// TIA Portal project "Clasificación, llenado y tapado de envases de pintura" (V16)

(* hardware
DEVICE "S7300/ET200M station_1"  S7-300 station
   slot 0: "Rail_0"  Rail  6ES7 390-1***0-0AA0
   slot 2: "PLC_1"  CPU 314C-2 PN/DP  6ES7 314-6EH04-0AB0  V3.3
      slot 2: "PROFINET interface_1"  PN-IO
         slot 1: "Port_1"  Port
         slot 2: "Port_2"  Port
      slot 5: "DI 24/DO 16_1"  DI24/DO16
      slot 6: "AI 5/AO 2_1"  AI5/AO2
      slot 7: "Count_1"  Counter
      slot 8: "Positioning_1"  Positioning
DEVICE "HMI_1"  TP700 Comfort
   slot 0: "HMI_1"  TP700 Comfort  6AV2 124-0GC01-0AX0  16.0.0.0
   slot 1: "HMI_RT_1"  TP700 Comfort  6AV2 124-0GC01-0AX0  16.0.0.0
   slot 5: "HMI_1.IE_CP_1"  PROFINET Interface  16.0.0.0
      slot 1: "Interfaz PROFINET_1"  PROFINET Interface
         slot 1: "Port_1"  Port
         slot 2: "Port_2"  Port
   slot 7: "HMI_1.MPI/DP_CP_1"  MPI/DP Interface  16.0.0.0
*)

// ===== PLC "PLC_1"  CPU 314C-2 PN/DP =====

VAR_GLOBAL   // PLC tag table "Entradas"
   "START" AT %I0.0 : Bool;
   "STOP" AT %I0.1 : Bool;
   "SPosIzq1" AT %I0.2 : Bool;
   "SPosDer1" AT %I0.3 : Bool;
   "PE" AT %I0.4 : Bool;
   "SVision" AT %ID30 : DInt;
   "SPosDer2" AT %I0.5 : Bool;
   "SPoseDer3" AT %I0.6 : Bool;
   "SPosIzq2" AT %I0.7 : Bool;
   "SPosIzq3" AT %I1.0 : Bool;
   "SEntrada" AT %I1.1 : Bool;
   "START_HMI" AT %M3.7 : Bool;
   "STOP_HMI" AT %M4.0 : Bool;
   "PE_HMI" AT %M4.1 : Bool;
   "EnvAzul" AT %M4.2 : Bool;
   "EnvVerde" AT %M4.3 : Bool;
   "SPosIzq4" AT %I1.2 : Bool;
   "SPosDer4" AT %I1.3 : Bool;
   "ContadorEnvAzul" AT %MW0 : Int;
   "ContadorEnvVerd" AT %MW2 : Int;
   "ClasificadorRecto" AT %M4.4 : Bool;
   "SEntTapaAzul" AT %I1.4 : Bool;
   "SEntTapaVerd" AT %I1.5 : Bool;
END_VAR

VAR_GLOBAL   // PLC tag table "Salidas"
   "FajaEntr" AT %Q0.0 : Bool;
   "ClasificadorGiro" AT %Q0.1 : Bool;
   "ClasificadorFaja+" AT %Q0.2 : Bool;
   "VLlenTanqIzq" AT %Q0.3 : Bool;
   "VLlenTanqDer" AT %Q0.4 : Bool;
   "FajaIzq1" AT %Q0.5 : Bool;
   "FajaIzq2" AT %Q0.6 : Bool;
   "FajaIzq3" AT %Q0.7 : Bool;
   "VLlenadoEnvIzq" AT %Q1.0 : Bool;
   "VDescTanqIzq" AT %Q1.1 : Bool;
   "FajaDer1" AT %Q1.2 : Bool;
   "VLlenadoEnvDer" AT %Q1.3 : Bool;
   "VDescTanqDer" AT %Q1.4 : Bool;
   "FajaDerecha2" AT %Q1.5 : Bool;
   "FajaDerecha3" AT %Q1.6 : Bool;
   "FajaIzq4" AT %Q1.7 : Bool;
   "FajaIzq5" AT %Q2.0 : Bool;
   "ClampDere1" AT %Q2.1 : Bool;
   "RaiseDere" AT %Q2.2 : Bool;
   "ClampDere2" AT %Q2.3 : Bool;
   "ClampIzq1" AT %Q2.4 : Bool;
   "RaiseIzq" AT %Q2.5 : Bool;
   "ClampIzq2" AT %Q2.6 : Bool;
   "MovZRDer" AT %Q2.7 : Bool;
   "MovXRder" AT %Q3.0 : Bool;
   "GrabRDer" AT %Q3.1 : Bool;
   "MovZRIzq" AT %Q3.2 : Bool;
   "MovXRizq" AT %Q3.3 : Bool;
   "GrabRIzq" AT %Q3.4 : Bool;
END_VAR

VAR_GLOBAL   // PLC tag table "Memorias"
   "Operativo" AT %M5.0 : Bool;
   "Tem1" AT %M0.1 : Bool;
   "Tem2" AT %M0.2 : Bool;
   "Tem3" AT %M0.3 : Bool;
   "Tem4" AT %M0.4 : Bool;
   "Tem6" AT %M0.6 : Bool;
   "Tem7" AT %M0.7 : Bool;
   "Tem8" AT %M1.0 : Bool;
   "Tem9" AT %M1.1 : Bool;
   "Tem10" AT %M1.2 : Bool;
   "Tem11" AT %M1.3 : Bool;
   "Tem12" AT %M1.4 : Bool;
   "Tem13" AT %M1.5 : Bool;
   "Tem14" AT %M1.6 : Bool;
   "Tem15" AT %M1.7 : Bool;
   "Tem16" AT %M2.0 : Bool;
   "Tem17" AT %M2.1 : Bool;
   "Tem18" AT %M2.2 : Bool;
   "Tem19" AT %M2.3 : Bool;
   "Tem20" AT %M2.4 : Bool;
   "Tem21" AT %M2.5 : Bool;
   "Tem22" AT %M2.6 : Bool;
   "Tem23" AT %M2.7 : Bool;
   "Tem24" AT %M3.0 : Bool;
   "Tem25" AT %M3.1 : Bool;
   "Tem26" AT %M3.2 : Bool;
   "Tem27" AT %M3.3 : Bool;
   "Tem28" AT %M3.4 : Bool;
   "Tem29" AT %M3.5 : Bool;
   "Tem30" AT %M3.6 : Bool;
END_VAR

DATA_BLOCK "Block_1_DB"   // DB1
{ S7_Optimized_Access := 'FALSE' }
VERSION : 0.1
// stored: InstanceOfName Block_1
"Block_1"
BEGIN
END_DATA_BLOCK

FUNCTION_BLOCK "Block_1"   // FB1, GRAPH
{ S7_Optimized_Access := 'FALSE' }
VERSION : 0.1
   VAR_INPUT
      OFF_SQ : Bool := false;   // Turn sequence off
      INIT_SQ : Bool := false;   // Set sequence to initial state
      ACK_EF : Bool := false;   // Acknowledge all errors and faults
      S_PREV : Bool := false;   // Output previous step in parameter S_NO
      S_NEXT : Bool := false;   // Indicate next step in parameter S_NO
      SW_AUTO : Bool := false;   // Automatic mode
      SW_TAP : Bool := false;   // Semiautomatic/switch with transition
      SW_TOP : Bool := false;   // Semiautomatic/ignore transition
      SW_MAN : Bool := false;   // Manual mode
      S_SEL : Int := 0;   // Select step to be output to S_NO
      S_ON : Bool := false;   // Activate step indicated in S_NO
      S_OFF : Bool := false;   // Deactivate step indicated S_NO
      T_PUSH : Bool := false;   // Enable transition to switch in semi automatic mode
   END_VAR
   VAR_OUTPUT
      S_NO : Int := 0;   // Step number
      S_MORE : Bool := false;   // More steps are available and can be shown in S_NO
      S_ACTIVE : Bool := false;   // Step indicated in S_NO is active
      ERR_FLT : Bool := false;   // Interlock or supervision group error
      AUTO_ON : Bool := false;   // Automatic mode is active
      TAP_ON : Bool := false;   // Semiautomatic mode/step with transition enabled
      TOP_ON : Bool := false;   // Semiautomatic mode/ignore transition enabled
      MAN_ON : Bool := false;   // Manual mode is active
   END_VAR
   VAR
      SWITCH : Array[0..2] of DWord;
      SW_SQTS : Array[0..36] of Byte;
      SW_ADDR : Word := 16#A;
      G7T_0 : GraphTransition;
      G7S_0 : GraphStep;
      PRE_CRIT : Array[0..0] of DWord;
      POST_CRIT : Array[0..0] of DWord;
      TVX : Array[0..8] of Byte;
      TTX : Array[0..8] of Byte;
      TSX : Array[0..6] of Byte;
      S00X : Array[0..6] of Byte;
      SOFFX : Array[0..6] of Byte;
      SONX : Array[0..6] of Byte;
      SAX : Array[0..6] of Byte;
      SERRX : Array[0..37] of Byte;
      SMX : Array[0..37] of Byte;
      S0X : Array[0..37] of Byte;
      S1X : Array[0..37] of Byte;
      S_DISPLAY : Int;   // Internal display of output parameter S_NO
      S_SEL_OLD : Int;   // Previous value in S_SEL
      S_DISPIDX : Byte;   // Index of the step in S_NO
      T_DISPIDX : Byte;   // Index of the transition displayed in T_NO
      MOPEDGE : Struct
         AUTO : Bool := false;
         MAN : Bool := false;
         TAP : Bool := false;
         TOP : Bool := false;
         ACK_S : Bool := false;
         REG_S : Bool := false;
         T_PREV : Bool := false;
         T_NEXT : Bool := false;
         LOCK : Bool := false;
         SUP : Bool := false;
         ACKREQ : Bool := false;
         SSKIP : Bool := false;
         OFF : Bool := false;
         INIT : Bool := false;
         HALT : Bool := false;
         TMS_HALT : Bool := false;
         OPS_ZERO : Bool := false;
         SACT_DISP : Bool := false;
         SEF_DISP : Bool := false;
         SALL_DISP : Bool := false;
         S_PREV : Bool := false;
         S_NEXT : Bool := false;
         S_SELOK : Bool := false;
         S_ON : Bool := false;
         S_OFF : Bool := false;
         T_PUSH : Bool := false;
         REG : Bool := false;
         ACK : Bool := false;
         IL_PERM : Bool := false;
         T_PERM : Bool := false;
         ILP_MAN : Bool := false;
      END_STRUCT;
      MOP : Struct   // Mode
         AUTO : Bool := true;   // Status: automatic mode
         MAN : Bool := false;   // Status: manual mode
         TAP : Bool := false;   // Status: semi automatic/switch with transition
         TOP : Bool := false;   // Status: semi automatic/ignore transition
         ACK_S : Bool := false;   // Request: acknowledge step at parameter S_NO
         REG_S : Bool := false;   // Request: register step indicated in S_NO
         T_PREV : Bool := false;   // Request: output previous valid transition in T_NO
         T_NEXT : Bool := false;   // Request: output next valid transition in T_NO
         LOCK : Bool := true;   // Status: interlocks activated
         SUP : Bool := true;   // Status: supervisions activated
         ACKREQ : Bool := true;   // Status: acknowledgment required
         SSKIP : Bool := false;   // Status: "Skip steps" enabled
         OFF : Bool := false;   // Request: deactivate all steps
         INIT : Bool := true;   // Request: set sequence to initial state
         HALT : Bool := false;   // Status: sequence halted
         TMS_HALT : Bool := false;   // Status: all internal timers held
         OPS_ZERO : Bool := false;   // Status: set all operands processed with N, L, D instructions to 0
         SACT_DISP : Bool := true;   // Status: display active steps only
         SEF_DISP : Bool := false;   // Status: display only steps with errors and disrupted steps
         SALL_DISP : Bool := false;   // Status: display all steps
         S_PREV : Bool := false;   // Request: output previous step to S_NO
         S_NEXT : Bool := false;   // Request: Output next step at S_NO parameter
         S_SELOK : Bool := false;   // Request: output step number from S_SEL to S_NO
         S_ON : Bool := false;   // Request: activate step indicated in S_NO
         S_OFF : Bool := false;   // Request: deactivate step at parameter S_NO
         T_PUSH : Bool := false;   // Request: transition switching enabled
         REG : Bool := false;   // Request: register all interlock and supervision errors
         ACK : Bool := false;   // Request: acknowledge all interlock and supervision errors
         IL_PERM : Bool := false;   // Status: permanent processing of all interlocks
         T_PERM : Bool := false;   // Status: permanent processing of all transitions
         ILP_MAN : Bool := false;   // Status: permanent processing of all interlocks in manual mode
      END_STRUCT;
      TICKS : Struct   // Clock speeds
         DELTA : Time := T#0ms;   // Time difference between cycles
         OLD : Time := T#0ms;   // 10 ms clock counter value in last cycle
         NEW : Time := T#0ms;   // 10 ms clock counter value in this cycle
      END_STRUCT;
      SQ_FLAGS : Struct   // Sequence bit memory
         ERR_FLT : Bool := false;   // Interlock and supervision group error
         ERROR : Bool := false;   // Interlock group error
         FAULT : Bool := false;   // Supervision group error
         RT_FAIL : Bool := false;   // Runtime error
         NO_SNO : Bool := false;   // Requested step number not found
         NF_OFL : Bool := false;   // Overflow: too many ON or OFF requests
         SA_OFL : Bool := false;   // Overflow: too many steps active
         TV_OFL : Bool := false;   // Overflow: too many valid transitions
         MSG_OFL : Bool := false;   // Overflow: not enough system resources for ALARM_S
         NO_SWI : Bool := false;   // Do not switch in this cycle
         CYC_OP : Bool := false;   // Cyclic execution of the sequence after initialization
         AS_MSG : Bool := true;   // Alarms during runtime enabled or disabled by instruction
         AS_SEND : Bool := false;   // Send alarms from WR_USMSG or only enter in diagnostics buffer
         SQ_BUSY : Bool := false;   // Internal edge memory bit for sequence processing
         SA_BUSY : Bool := false;   // Internal edge memory bit for sequence processing
         AS_SIG : Bool := false;   // Edge memory bit for alarms from Alarm_S and Alarm_SQ
      END_STRUCT;
      S_PTR : DWord := 16#13F0;
      S_PTR2 : DWord := 16#0;
      S_PTR3 : DWord := 16#3EA0;
      S_PTR4 : DWord := 16#3D70;
      T_PTR : DWord := 16#3C40;
      C_AR2 : DWord := 16#0;
      M_FBDB : DWord := 16#10000;
      M_SNO : Word := 16#0;
      M_EVID : Word := 16#0;
      M_EVIL : C_Alarm_s;
      M_EVSV : C_Alarm_s;
      M_EV : DWord := 16#3A50;
      CRIT : Array[0..31] of Bool;
      S_START : Byte := 16#0;
      S_IDX : Byte := 16#0;
      S_INT : Int := 72;
      S_TMP : Byte := 16#0;
      T_START : Byte := 16#0;
      T_IDX : Byte := 16#0;
      T_TMP : Byte := 16#0;
      T_TMP2 : Byte := 16#00;
      TV_POT : Byte := 16#06;
      RETURN1 : Byte := 16#0;
      RETURN2 : Byte := 16#0;
      SINI : Array[0..6] of Byte;
      LSTT : Array[0..35] of Byte;
      ATAJ : Array[0..35] of Byte;
      ATAB : Array[0..35] of Byte;
      PSTT : Array[0..35] of Byte;
      NSTT : Array[0..35] of Byte;
      ASSJ : Array[0..36] of Byte;
      ASSB : Array[0..36] of Byte;
      PTTS : Array[0..36] of Byte;
      NTTS : Array[0..36] of Byte;
      PRE_CNT : Word := 16#1;
      POST_CNT : Word := 16#1;
      ADR_COND : Word := 16#0;
      MAX_TVAL : Byte := 16#7;
      MAX_SACT : Byte := 16#5;
      MAX_CRIT : Byte := 16#4;
      T_CNT : Byte := 16#23;
      SUP_CNT : Byte := 16#0;
      LOCK_CNT : Byte := 16#0;
      S_CNT : Byte := 16#24;
      SQ_CNT : Byte := 16#1;
      PRS_INPAR : DWord := 16#E000FEC8;
      PRS_OUTPAR : DWord := 16#E000800F;
      GC_FLAGS : Struct
         T_MACH : Byte := 16#EB;
         COND_ED : Byte := 16#E3;
         W_LEVEL : Byte := 16#D5;
         FB_IF : Byte := 16#FA;
         AS_MSG : Word := 16#404;
         SSB : Word := 16#108;
         DILG : Word := 16#9CE;
         ADDR_T0 : Word := 16#3E;
         CRIT_AVAIL : Bool := false;
         SSKIP_AVAIL : Bool := true;
         SSKIP_ON : Bool := false;
         ACK_REQ : Bool := true;
         SYNC_AVAIL : Bool := true;
         ILP_MAN : Bool := false;
         SWM_LOCKED : Bool := false;
         SAVE_SW : Bool := true;
      END_STRUCT;
      G7_FBMARK : Byte := 16#3C;
      G7_RELEASE : Byte := 16#3C;
      G7_ID2 : Byte := 16#37;
      G7_ID1 : Byte := 16#47;
   END_VAR
   // SWITCH[0] := 16#2020;
   // SWITCH[1] := 16#20;
   // SWITCH[2] := 16#20000000;
   // SW_SQTS[0] := 16#9;
   // SW_SQTS[4] := 16#1;
   // SW_SQTS[5] := 16#1;
   // SW_SQTS[6] := 16#1;
   // SW_SQTS[7] := 16#1;
   // SW_SQTS[8] := 16#2;
   // SW_SQTS[9] := 16#3;
   // SW_SQTS[10] := 16#2;
   // SW_SQTS[11] := 16#2;
   // SW_SQTS[12] := 16#2;
   // SW_SQTS[13] := 16#2;
   // SW_SQTS[14] := 16#2;
   // SW_SQTS[15] := 16#2;
   // SW_SQTS[16] := 16#2;
   // SW_SQTS[17] := 16#3;
   // SW_SQTS[18] := 16#4;
   // SW_SQTS[19] := 16#5;
   // SW_SQTS[20] := 16#5;
   // SW_SQTS[21] := 16#5;
   // SW_SQTS[22] := 16#5;
   // SW_SQTS[23] := 16#5;
   // SW_SQTS[24] := 16#5;
   // SW_SQTS[25] := 16#6;
   // SW_SQTS[26] := 16#7;
   // SW_SQTS[27] := 16#7;
   // SW_SQTS[28] := 16#6;
   // SW_SQTS[29] := 16#6;
   // SW_SQTS[30] := 16#6;
   // SW_SQTS[31] := 16#6;
   // SW_SQTS[32] := 16#6;
   // SW_SQTS[33] := 16#6;
   // SW_SQTS[34] := 16#6;
   // SW_SQTS[35] := 16#8;
   // SW_SQTS[36] := 16#1;
   // TVX[0] := 16#1;
   // TTX[0] := 16#1;
   // TSX[0] := 16#1;
   // S00X[0] := 16#1;
   // SOFFX[0] := 16#1;
   // SONX[0] := 16#1;
   // SAX[0] := 16#1;
   // SERRX[0] := 16#1;
   // SMX[0] := 16#1;
   // S0X[0] := 16#1;
   // S1X[0] := 16#1;
   // SINI[0] := 16#2;
   // SINI[1] := 16#1;
   // SINI[2] := 0;
   // SINI[3] := 0;
   // SINI[4] := 0;
   // SINI[5] := 0;
   // SINI[6] := 0;
   // LSTT[0] := 0;
   // LSTT[1] := 0;
   // LSTT[2] := 0;
   // LSTT[3] := 0;
   // LSTT[4] := 0;
   // LSTT[5] := 0;
   // LSTT[6] := 0;
   // LSTT[7] := 0;
   // LSTT[8] := 0;
   // LSTT[9] := 0;
   // LSTT[10] := 0;
   // LSTT[11] := 0;
   // LSTT[12] := 0;
   // LSTT[13] := 0;
   // LSTT[14] := 0;
   // LSTT[15] := 0;
   // LSTT[16] := 0;
   // LSTT[17] := 0;
   // LSTT[18] := 0;
   // LSTT[19] := 16#1;
   // LSTT[20] := 0;
   // LSTT[21] := 0;
   // LSTT[22] := 0;
   // LSTT[23] := 0;
   // LSTT[24] := 0;
   // LSTT[25] := 0;
   // LSTT[26] := 0;
   // LSTT[27] := 0;
   // LSTT[28] := 0;
   // LSTT[29] := 0;
   // LSTT[30] := 0;
   // LSTT[31] := 0;
   // LSTT[32] := 0;
   // LSTT[33] := 0;
   // LSTT[34] := 0;
   // LSTT[35] := 16#1;
   // ATAJ[0] := 0;
   // ATAJ[1] := 16#1;
   // ATAJ[2] := 16#2;
   // ATAJ[3] := 16#3;
   // ATAJ[4] := 16#4;
   // ATAJ[5] := 16#5;
   // ATAJ[6] := 16#6;
   // ATAJ[7] := 16#7;
   // ATAJ[8] := 16#8;
   // ATAJ[9] := 16#9;
   // ATAJ[10] := 16#A;
   // ATAJ[11] := 16#B;
   // ATAJ[12] := 16#C;
   // ATAJ[13] := 16#D;
   // ATAJ[14] := 16#E;
   // ATAJ[15] := 16#F;
   // ATAJ[16] := 16#10;
   // ATAJ[17] := 16#11;
   // ATAJ[18] := 16#12;
   // ATAJ[19] := 16#13;
   // ATAJ[20] := 16#14;
   // ATAJ[21] := 16#15;
   // ATAJ[22] := 16#16;
   // ATAJ[23] := 16#17;
   // ATAJ[24] := 16#18;
   // ATAJ[25] := 16#19;
   // ATAJ[26] := 16#1A;
   // ATAJ[27] := 16#1B;
   // ATAJ[28] := 16#1C;
   // ATAJ[29] := 16#1D;
   // ATAJ[30] := 16#1E;
   // ATAJ[31] := 16#1F;
   // ATAJ[32] := 16#20;
   // ATAJ[33] := 16#21;
   // ATAJ[34] := 16#22;
   // ATAJ[35] := 16#23;
   // ATAB[0] := 0;
   // ATAB[1] := 16#1;
   // ATAB[2] := 16#2;
   // ATAB[3] := 16#4;
   // ATAB[4] := 16#3;
   // ATAB[5] := 16#5;
   // ATAB[6] := 16#6;
   // ATAB[7] := 16#7;
   // ATAB[8] := 16#8;
   // ATAB[9] := 16#9;
   // ATAB[10] := 16#A;
   // ATAB[11] := 16#B;
   // ATAB[12] := 16#C;
   // ATAB[13] := 16#D;
   // ATAB[14] := 16#E;
   // ATAB[15] := 16#F;
   // ATAB[16] := 16#10;
   // ATAB[17] := 16#11;
   // ATAB[18] := 16#12;
   // ATAB[19] := 16#13;
   // ATAB[20] := 16#14;
   // ATAB[21] := 16#15;
   // ATAB[22] := 16#16;
   // ATAB[23] := 16#17;
   // ATAB[24] := 16#18;
   // ATAB[25] := 16#19;
   // ATAB[26] := 16#1A;
   // ATAB[27] := 16#1B;
   // ATAB[28] := 16#1C;
   // ATAB[29] := 16#1D;
   // ATAB[30] := 16#1E;
   // ATAB[31] := 16#1F;
   // ATAB[32] := 16#20;
   // ATAB[33] := 16#21;
   // ATAB[34] := 16#22;
   // ATAB[35] := 16#23;
   // PSTT[0] := 0;
   // PSTT[1] := 16#1;
   // PSTT[2] := 16#2;
   // PSTT[3] := 16#3;
   // PSTT[4] := 16#3;
   // PSTT[5] := 16#4;
   // PSTT[6] := 16#5;
   // PSTT[7] := 16#6;
   // PSTT[8] := 16#7;
   // PSTT[9] := 16#24;
   // PSTT[10] := 16#9;
   // PSTT[11] := 16#8;
   // PSTT[12] := 16#A;
   // PSTT[13] := 16#B;
   // PSTT[14] := 16#C;
   // PSTT[15] := 16#D;
   // PSTT[16] := 16#E;
   // PSTT[17] := 16#F;
   // PSTT[18] := 16#11;
   // PSTT[19] := 16#12;
   // PSTT[20] := 16#13;
   // PSTT[21] := 16#14;
   // PSTT[22] := 16#15;
   // PSTT[23] := 16#16;
   // PSTT[24] := 16#17;
   // PSTT[25] := 16#18;
   // PSTT[26] := 16#1A;
   // PSTT[27] := 16#19;
   // PSTT[28] := 16#1C;
   // PSTT[29] := 16#1D;
   // PSTT[30] := 16#1E;
   // PSTT[31] := 16#1F;
   // PSTT[32] := 16#20;
   // PSTT[33] := 16#21;
   // PSTT[34] := 16#1B;
   // PSTT[35] := 16#23;
   // NSTT[0] := 16#1;
   // NSTT[1] := 16#2;
   // NSTT[2] := 16#3;
   // NSTT[3] := 16#13;
   // NSTT[4] := 16#4;
   // NSTT[5] := 16#5;
   // NSTT[6] := 16#6;
   // NSTT[7] := 16#7;
   // NSTT[8] := 16#24;
   // NSTT[9] := 16#9;
   // NSTT[10] := 16#11;
   // NSTT[11] := 16#A;
   // NSTT[12] := 16#B;
   // NSTT[13] := 16#C;
   // NSTT[14] := 16#D;
   // NSTT[15] := 16#E;
   // NSTT[16] := 16#F;
   // NSTT[17] := 16#10;
   // NSTT[18] := 16#12;
   // NSTT[19] := 16#1;
   // NSTT[20] := 16#14;
   // NSTT[21] := 16#15;
   // NSTT[22] := 16#16;
   // NSTT[23] := 16#17;
   // NSTT[24] := 16#18;
   // NSTT[25] := 16#1A;
   // NSTT[26] := 16#1B;
   // NSTT[27] := 16#1C;
   // NSTT[28] := 16#1D;
   // NSTT[29] := 16#1E;
   // NSTT[30] := 16#1F;
   // NSTT[31] := 16#20;
   // NSTT[32] := 16#21;
   // NSTT[33] := 16#22;
   // NSTT[34] := 16#23;
   // NSTT[35] := 16#1;
   // ASSJ[0] := 0;
   // ASSJ[1] := 16#1;
   // ASSJ[2] := 16#2;
   // ASSJ[3] := 16#3;
   // ASSJ[4] := 16#4;
   // ASSJ[5] := 16#5;
   // ASSJ[6] := 16#6;
   // ASSJ[7] := 16#7;
   // ASSJ[8] := 16#8;
   // ASSJ[9] := 16#9;
   // ASSJ[10] := 16#A;
   // ASSJ[11] := 16#B;
   // ASSJ[12] := 16#C;
   // ASSJ[13] := 16#D;
   // ASSJ[14] := 16#E;
   // ASSJ[15] := 16#F;
   // ASSJ[16] := 16#11;
   // ASSJ[17] := 16#10;
   // ASSJ[18] := 16#12;
   // ASSJ[19] := 16#13;
   // ASSJ[20] := 16#14;
   // ASSJ[21] := 16#15;
   // ASSJ[22] := 16#16;
   // ASSJ[23] := 16#17;
   // ASSJ[24] := 16#18;
   // ASSJ[25] := 16#19;
   // ASSJ[26] := 16#1A;
   // ASSJ[27] := 16#22;
   // ASSJ[28] := 16#1C;
   // ASSJ[29] := 16#1D;
   // ASSJ[30] := 16#1E;
   // ASSJ[31] := 16#1F;
   // ASSJ[32] := 16#20;
   // ASSJ[33] := 16#21;
   // ASSJ[34] := 16#1B;
   // ASSJ[35] := 16#23;
   // ASSJ[36] := 16#24;
   // ASSB[0] := 0;
   // ASSB[1] := 16#1;
   // ASSB[2] := 16#2;
   // ASSB[3] := 16#3;
   // ASSB[4] := 16#4;
   // ASSB[5] := 16#5;
   // ASSB[6] := 16#6;
   // ASSB[7] := 16#7;
   // ASSB[8] := 16#9;
   // ASSB[9] := 16#8;
   // ASSB[10] := 16#A;
   // ASSB[11] := 16#B;
   // ASSB[12] := 16#C;
   // ASSB[13] := 16#D;
   // ASSB[14] := 16#E;
   // ASSB[15] := 16#F;
   // ASSB[16] := 16#10;
   // ASSB[17] := 16#11;
   // ASSB[18] := 16#12;
   // ASSB[19] := 16#13;
   // ASSB[20] := 16#14;
   // ASSB[21] := 16#15;
   // ASSB[22] := 16#16;
   // ASSB[23] := 16#17;
   // ASSB[24] := 16#18;
   // ASSB[25] := 16#1A;
   // ASSB[26] := 16#19;
   // ASSB[27] := 16#1B;
   // ASSB[28] := 16#1C;
   // ASSB[29] := 16#1D;
   // ASSB[30] := 16#1E;
   // ASSB[31] := 16#1F;
   // ASSB[32] := 16#20;
   // ASSB[33] := 16#21;
   // ASSB[34] := 16#22;
   // ASSB[35] := 16#23;
   // ASSB[36] := 16#24;
   // PTTS[0] := 0;
   // PTTS[2] := 16#1;
   // PTTS[3] := 16#2;
   // PTTS[4] := 16#4;
   // PTTS[5] := 16#5;
   // PTTS[6] := 16#6;
   // PTTS[7] := 16#7;
   // PTTS[8] := 16#9;
   // PTTS[9] := 16#9;
   // PTTS[10] := 16#B;
   // PTTS[11] := 16#C;
   // PTTS[12] := 16#D;
   // PTTS[13] := 16#E;
   // PTTS[14] := 16#F;
   // PTTS[15] := 16#10;
   // PTTS[16] := 16#11;
   // PTTS[17] := 16#A;
   // PTTS[18] := 16#12;
   // PTTS[19] := 16#3;
   // PTTS[20] := 16#14;
   // PTTS[21] := 16#15;
   // PTTS[22] := 16#16;
   // PTTS[23] := 16#17;
   // PTTS[24] := 16#18;
   // PTTS[25] := 16#19;
   // PTTS[26] := 16#19;
   // PTTS[27] := 16#1A;
   // PTTS[28] := 16#1B;
   // PTTS[29] := 16#1C;
   // PTTS[30] := 16#1D;
   // PTTS[31] := 16#1E;
   // PTTS[32] := 16#1F;
   // PTTS[33] := 16#20;
   // PTTS[34] := 16#21;
   // PTTS[35] := 16#22;
   // PTTS[36] := 16#8;
   // NTTS[0] := 0;
   // NTTS[1] := 16#1;
   // NTTS[2] := 16#2;
   // NTTS[3] := 16#4;
   // NTTS[4] := 16#5;
   // NTTS[5] := 16#6;
   // NTTS[6] := 16#7;
   // NTTS[7] := 16#8;
   // NTTS[8] := 16#B;
   // NTTS[9] := 16#A;
   // NTTS[10] := 16#C;
   // NTTS[11] := 16#D;
   // NTTS[12] := 16#E;
   // NTTS[13] := 16#F;
   // NTTS[14] := 16#10;
   // NTTS[15] := 16#11;
   // NTTS[16] := 16#12;
   // NTTS[17] := 16#12;
   // NTTS[18] := 16#13;
   // NTTS[19] := 16#14;
   // NTTS[20] := 16#15;
   // NTTS[21] := 16#16;
   // NTTS[22] := 16#17;
   // NTTS[23] := 16#18;
   // NTTS[24] := 16#19;
   // NTTS[25] := 16#1B;
   // NTTS[26] := 16#1A;
   // NTTS[27] := 16#22;
   // NTTS[28] := 16#1C;
   // NTTS[29] := 16#1D;
   // NTTS[30] := 16#1E;
   // NTTS[31] := 16#1F;
   // NTTS[32] := 16#20;
   // NTTS[33] := 16#21;
   // NTTS[34] := 16#22;
   // NTTS[35] := 16#23;
   // NTTS[36] := 16#9;
BEGIN
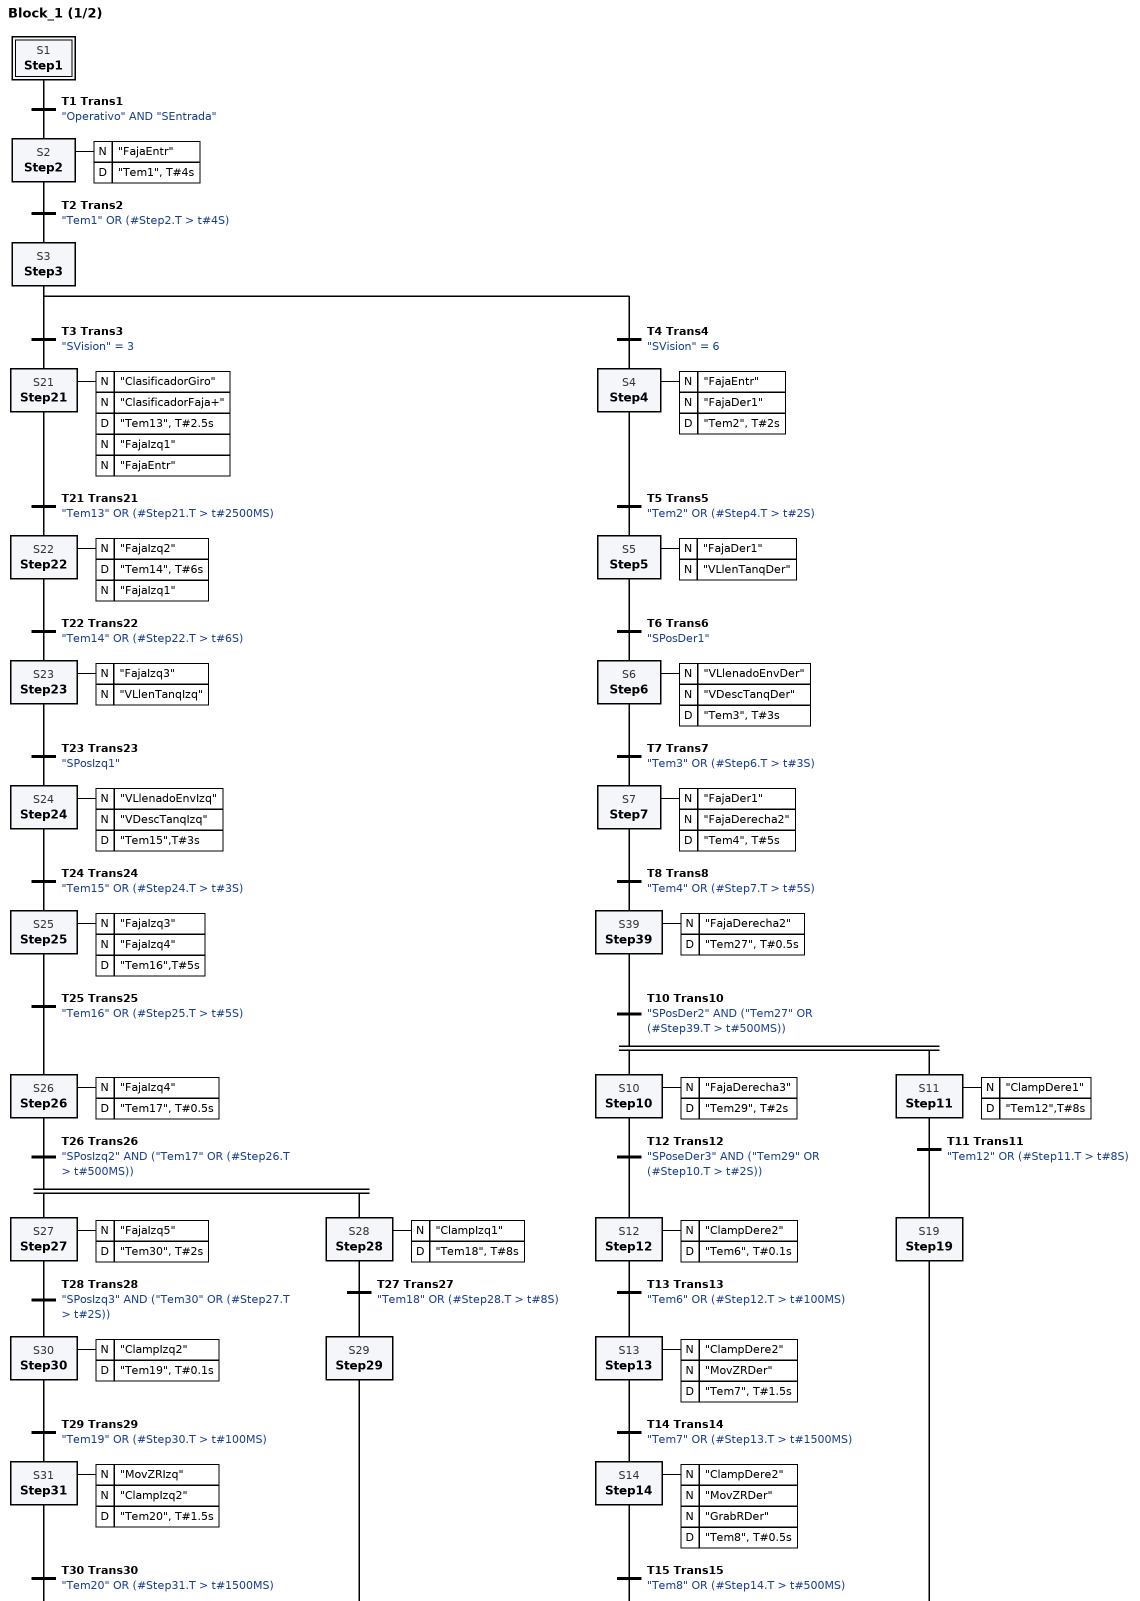
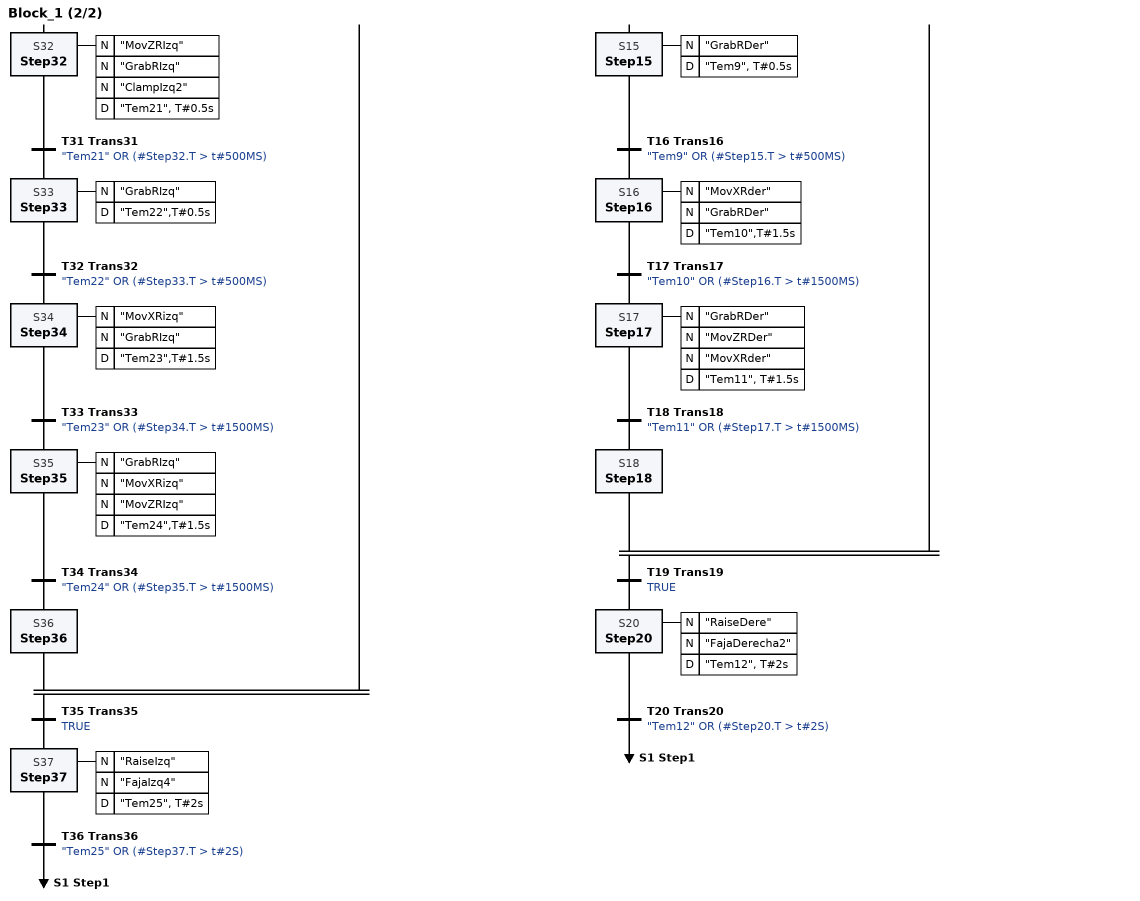
   // sequencer 1
   INITIAL_STEP Step1:   // S1
   END_STEP
   TRANSITION Trans1 FROM Step1 TO Step2   // T1
      := "Operativo" AND "SEntrada";
   END_TRANSITION
   STEP Step2:   // S2
              N    "FajaEntr"
              D    "Tem1", T#4s
   END_STEP
   TRANSITION Trans2 FROM Step2 TO Step3   // T2
      := "Tem1" OR (#Step2.T > t#4S);
   END_TRANSITION
   STEP Step3:   // S3
   END_STEP
   TRANSITION Trans3 FROM Step3 TO Step21   // T3
      := "SVision" = 3;
   END_TRANSITION
   TRANSITION Trans4 FROM Step3 TO Step4   // T4
      := "SVision" = 6;
   END_TRANSITION
   STEP Step4:   // S4
              N    "FajaEntr"
              N    "FajaDer1"
              D    "Tem2", T#2s
   END_STEP
   TRANSITION Trans5 FROM Step4 TO Step5   // T5
      := "Tem2" OR (#Step4.T > t#2S);
   END_TRANSITION
   STEP Step5:   // S5
              N    "FajaDer1"
              N    "VLlenTanqDer"
   END_STEP
   TRANSITION Trans6 FROM Step5 TO Step6   // T6
      := "SPosDer1";
   END_TRANSITION
   STEP Step6:   // S6
              N    "VLlenadoEnvDer"
              N    "VDescTanqDer"
              D    "Tem3", T#3s
   END_STEP
   TRANSITION Trans7 FROM Step6 TO Step7   // T7
      := "Tem3" OR (#Step6.T > t#3S);
   END_TRANSITION
   STEP Step7:   // S7
              N    "FajaDer1"
              N    "FajaDerecha2"
              D    "Tem4", T#5s
   END_STEP
   TRANSITION Trans8 FROM Step7 TO Step39   // T8
      := "Tem4" OR (#Step7.T > t#5S);
   END_TRANSITION
   STEP Step39:   // S39
              N    "FajaDerecha2"
              D    "Tem27", T#0.5s
   END_STEP
   TRANSITION Trans10 FROM Step39 TO (Step10, Step11)   // T10
      := "SPosDer2" AND ("Tem27" OR (#Step39.T > t#500MS));
   END_TRANSITION
   STEP Step10:   // S10
              N    "FajaDerecha3"
              D    "Tem29", T#2s
   END_STEP
   TRANSITION Trans12 FROM Step10 TO Step12   // T12
      := "SPoseDer3" AND ("Tem29" OR (#Step10.T > t#2S));
   END_TRANSITION
   STEP Step11:   // S11
              N    "ClampDere1"
              D    "Tem12",T#8s
   END_STEP
   TRANSITION Trans11 FROM Step11 TO Step19   // T11
      := "Tem12" OR (#Step11.T > t#8S);
   END_TRANSITION
   STEP Step12:   // S12
              N    "ClampDere2"
              D    "Tem6", T#0.1s
   END_STEP
   TRANSITION Trans13 FROM Step12 TO Step13   // T13
      := "Tem6" OR (#Step12.T > t#100MS);
   END_TRANSITION
   STEP Step13:   // S13
              N    "ClampDere2"
              N    "MovZRDer"
              D    "Tem7", T#1.5s
   END_STEP
   TRANSITION Trans14 FROM Step13 TO Step14   // T14
      := "Tem7" OR (#Step13.T > t#1500MS);
   END_TRANSITION
   STEP Step14:   // S14
              N    "ClampDere2"
              N    "MovZRDer"
              N    "GrabRDer"
              D    "Tem8", T#0.5s
   END_STEP
   TRANSITION Trans15 FROM Step14 TO Step15   // T15
      := "Tem8" OR (#Step14.T > t#500MS);
   END_TRANSITION
   STEP Step15:   // S15
              N    "GrabRDer"
              D    "Tem9", T#0.5s
   END_STEP
   TRANSITION Trans16 FROM Step15 TO Step16   // T16
      := "Tem9" OR (#Step15.T > t#500MS);
   END_TRANSITION
   STEP Step16:   // S16
              N    "MovXRder"
              N    "GrabRDer"
              D    "Tem10",T#1.5s
   END_STEP
   TRANSITION Trans17 FROM Step16 TO Step17   // T17
      := "Tem10" OR (#Step16.T > t#1500MS);
   END_TRANSITION
   STEP Step17:   // S17
              N    "GrabRDer"
              N    "MovZRDer"
              N    "MovXRder"
              D    "Tem11", T#1.5s
   END_STEP
   TRANSITION Trans18 FROM Step17 TO Step18   // T18
      := "Tem11" OR (#Step17.T > t#1500MS);
   END_TRANSITION
   STEP Step18:   // S18
   END_STEP
   TRANSITION Trans19 FROM (Step19, Step18) TO Step20   // T19
      := TRUE;
   END_TRANSITION
   STEP Step19:   // S19
   END_STEP
   STEP Step20:   // S20
              N    "RaiseDere"
              N    "FajaDerecha2"
              D    "Tem12", T#2s
   END_STEP
   TRANSITION Trans20 FROM Step20 TO Step1   // T20, jump
      := "Tem12" OR (#Step20.T > t#2S);
   END_TRANSITION
   STEP Step21:   // S21
              N    "ClasificadorGiro"
              N    "ClasificadorFaja+"
              D    "Tem13", T#2.5s
              N    "FajaIzq1"
              N    "FajaEntr"
   END_STEP
   TRANSITION Trans21 FROM Step21 TO Step22   // T21
      := "Tem13" OR (#Step21.T > t#2500MS);
   END_TRANSITION
   STEP Step22:   // S22
              N    "FajaIzq2"
              D    "Tem14", T#6s
              N    "FajaIzq1"
   END_STEP
   TRANSITION Trans22 FROM Step22 TO Step23   // T22
      := "Tem14" OR (#Step22.T > t#6S);
   END_TRANSITION
   STEP Step23:   // S23
              N    "FajaIzq3"
              N    "VLlenTanqIzq"
   END_STEP
   TRANSITION Trans23 FROM Step23 TO Step24   // T23
      := "SPosIzq1";
   END_TRANSITION
   STEP Step24:   // S24
              N    "VLlenadoEnvIzq"
              N    "VDescTanqIzq"
              D    "Tem15",T#3s
   END_STEP
   TRANSITION Trans24 FROM Step24 TO Step25   // T24
      := "Tem15" OR (#Step24.T > t#3S);
   END_TRANSITION
   STEP Step25:   // S25
              N    "FajaIzq3"
              N    "FajaIzq4"
              D    "Tem16",T#5s
   END_STEP
   TRANSITION Trans25 FROM Step25 TO Step26   // T25
      := "Tem16" OR (#Step25.T > t#5S);
   END_TRANSITION
   STEP Step26:   // S26
              N    "FajaIzq4"
              D    "Tem17", T#0.5s
   END_STEP
   TRANSITION Trans26 FROM Step26 TO (Step27, Step28)   // T26
      := "SPosIzq2" AND ("Tem17" OR (#Step26.T > t#500MS));
   END_TRANSITION
   STEP Step27:   // S27
              N    "FajaIzq5"
              D    "Tem30", T#2s
   END_STEP
   TRANSITION Trans28 FROM Step27 TO Step30   // T28
      := "SPosIzq3" AND ("Tem30" OR (#Step27.T > t#2S));
   END_TRANSITION
   STEP Step28:   // S28
              N    "ClampIzq1"
              D    "Tem18", T#8s
   END_STEP
   TRANSITION Trans27 FROM Step28 TO Step29   // T27
      := "Tem18" OR (#Step28.T > t#8S);
   END_TRANSITION
   STEP Step29:   // S29
   END_STEP
   STEP Step30:   // S30
              N    "ClampIzq2"
              D    "Tem19", T#0.1s
   END_STEP
   TRANSITION Trans29 FROM Step30 TO Step31   // T29
      := "Tem19" OR (#Step30.T > t#100MS);
   END_TRANSITION
   STEP Step31:   // S31
              N    "MovZRIzq"
              N    "ClampIzq2"
              D    "Tem20", T#1.5s
   END_STEP
   TRANSITION Trans30 FROM Step31 TO Step32   // T30
      := "Tem20" OR (#Step31.T > t#1500MS);
   END_TRANSITION
   STEP Step32:   // S32
              N    "MovZRIzq"
              N    "GrabRIzq"
              N    "ClampIzq2"
              D    "Tem21", T#0.5s
   END_STEP
   TRANSITION Trans31 FROM Step32 TO Step33   // T31
      := "Tem21" OR (#Step32.T > t#500MS);
   END_TRANSITION
   STEP Step33:   // S33
              N    "GrabRIzq"
              D    "Tem22",T#0.5s
   END_STEP
   TRANSITION Trans32 FROM Step33 TO Step34   // T32
      := "Tem22" OR (#Step33.T > t#500MS);
   END_TRANSITION
   STEP Step34:   // S34
              N    "MovXRizq"
              N    "GrabRIzq"
              D    "Tem23",T#1.5s
   END_STEP
   TRANSITION Trans33 FROM Step34 TO Step35   // T33
      := "Tem23" OR (#Step34.T > t#1500MS);
   END_TRANSITION
   STEP Step35:   // S35
              N    "GrabRIzq"
              N    "MovXRizq"
              N    "MovZRIzq"
              D    "Tem24",T#1.5s
   END_STEP
   TRANSITION Trans34 FROM Step35 TO Step36   // T34
      := "Tem24" OR (#Step35.T > t#1500MS);
   END_TRANSITION
   STEP Step36:   // S36
   END_STEP
   TRANSITION Trans35 FROM (Step29, Step36) TO Step37   // T35
      := TRUE;
   END_TRANSITION
   STEP Step37:   // S37
              N    "RaiseIzq"
              N    "FajaIzq4"
              D    "Tem25", T#2s
   END_STEP
   TRANSITION Trans36 FROM Step37 TO Step1   // T36, jump
      := "Tem25" OR (#Step37.T > t#2S);
   END_TRANSITION
END_FUNCTION_BLOCK

ORGANIZATION_BLOCK "Main"   // OB1, LAD
TITLE = "Main Program Sweep (Cycle)"
{ S7_Optimized_Access := 'FALSE' }
VERSION : 0.1
   VAR_TEMP
      OB1_EV_CLASS : Byte;   // Bits 0-3 = 1 (Coming event), Bits 4-7 = 1 (Event class 1)
      OB1_SCAN_1 : Byte;   // 1 (Cold restart scan 1 of OB 1), 3 (Scan 2-n of OB 1)
      OB1_PRIORITY : Byte;   // Priority of OB Execution
      OB1_OB_NUMBR : Byte;   // 1 (Organization block 1, OB1)
      OB1_RESERVED_1 : Byte;   // Reserved for system
      OB1_RESERVED_2 : Byte;   // Reserved for system
      OB1_PREV_CYCLE : Int;   // Cycle time of previous OB1 scan (milliseconds)
      OB1_MIN_CYCLE : Int;   // Minimum cycle time of OB1 (milliseconds)
      OB1_MAX_CYCLE : Int;   // Maximum cycle time of OB1 (milliseconds)
      OB1_DATE_TIME : Date_And_Time;   // Date and time OB1 started
   END_VAR
BEGIN

REGION Network 1
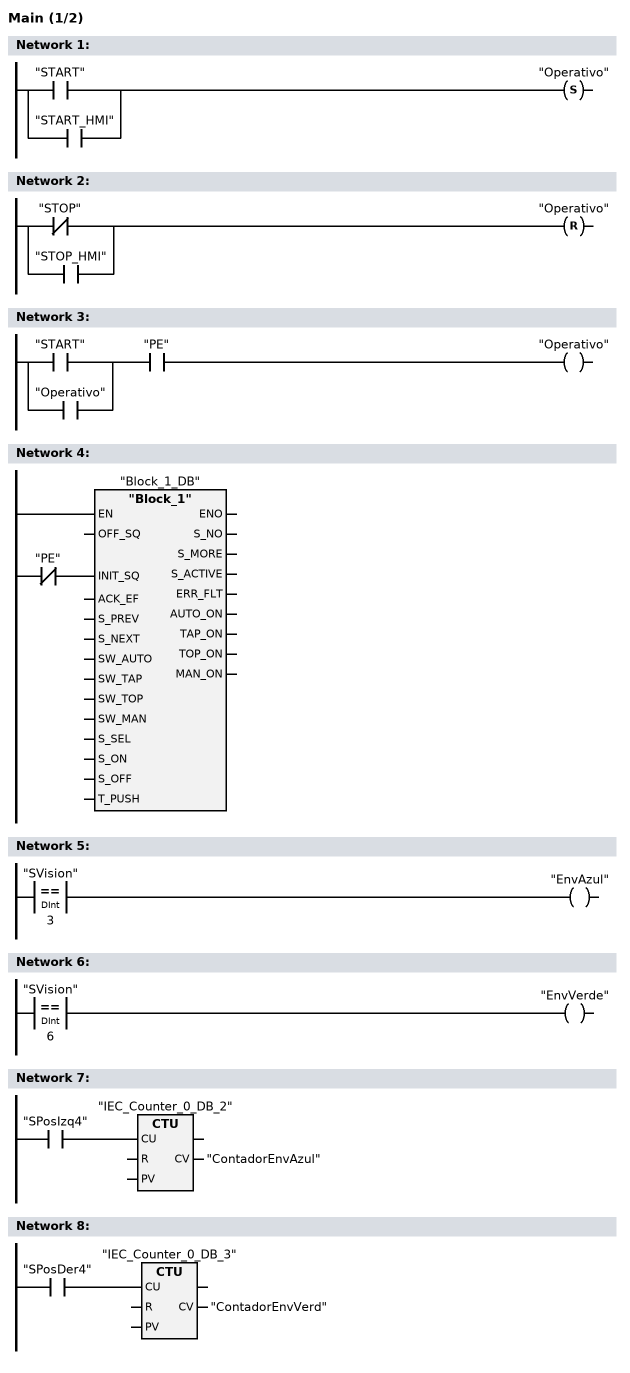
   RUNG wire#powerrail
      Contact( "START" )
      wire#w1
      S_Coil( "Operativo" )
   END_RUNG
   RUNG wire#powerrail
      Contact( "START_HMI" )
   END_RUNG wire#w1
   // the same network as SCL:
   IF "START" OR "START_HMI" THEN "Operativo" := TRUE; END_IF;
END_REGION

REGION Network 2
   RUNG wire#powerrail
      I_Contact( "STOP" )
      wire#w1
      R_Coil( "Operativo" )
   END_RUNG
   RUNG wire#powerrail
      Contact( "STOP_HMI" )
   END_RUNG wire#w1
   // the same network as SCL:
   IF NOT "STOP" OR "STOP_HMI" THEN "Operativo" := FALSE; END_IF;
END_REGION

REGION Network 3
   RUNG wire#powerrail
      Contact( "START" )
      wire#w1
      Contact( "PE" )
      Coil( "Operativo" )
   END_RUNG
   RUNG wire#powerrail
      Contact( "Operativo" )
   END_RUNG wire#w1
   // the same network as SCL:
   "Operativo" := ("START" OR "Operativo") AND "PE";
END_REGION

REGION Network 4
   RUNG wire#powerrail
      "Block_1_DB"(INIT_SQ := wire#w1, OFF_SQ :=, ACK_EF :=, S_PREV :=, S_NEXT :=, SW_AUTO :=, SW_TAP :=, SW_TOP :=, SW_MAN :=, S_SEL :=, S_ON :=, S_OFF :=, T_PUSH :=, S_NO =>, S_MORE =>, S_ACTIVE =>, ERR_FLT =>, AUTO_ON =>, TAP_ON =>, TOP_ON =>, MAN_ON =>)
   END_RUNG
   RUNG wire#powerrail
      I_Contact( "PE" )
   END_RUNG wire#w1
   // the same network as SCL:
   "Block_1_DB"(INIT_SQ := NOT "PE");   // "Block_1"
END_REGION

REGION Network 5
   RUNG wire#powerrail
      { S7_Templates := "SrcType := DInt" } EQ_Contact(in1 := "SVision", in2 := 3)
      Coil( "EnvAzul" )
   END_RUNG
   // the same network as SCL:
   "EnvAzul" := "SVision" = 3;
END_REGION

REGION Network 6
   RUNG wire#powerrail
      { S7_Templates := "SrcType := DInt" } EQ_Contact(in1 := "SVision", in2 := 6)
      Coil( "EnvVerde" )
   END_RUNG
   // the same network as SCL:
   "EnvVerde" := "SVision" = 6;
END_REGION

REGION Network 7
   "IEC_Counter_0_DB_2".CTU(CU := "SPosIzq4", CV => "ContadorEnvAzul");
END_REGION

REGION Network 8
   "IEC_Counter_0_DB_3".CTU(CU := "SPosDer4", CV => "ContadorEnvVerd");
END_REGION

REGION Network 9
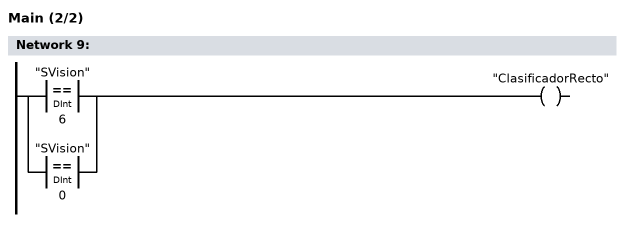
   RUNG wire#powerrail
      { S7_Templates := "SrcType := DInt" } EQ_Contact(in1 := "SVision", in2 := 6)
      wire#w1
      Coil( "ClasificadorRecto" )
   END_RUNG
   RUNG wire#powerrail
      { S7_Templates := "SrcType := DInt" } EQ_Contact(in1 := "SVision", in2 := 0)
   END_RUNG wire#w1
   // the same network as SCL:
   "ClasificadorRecto" := ("SVision" = 6) OR ("SVision" = 0);
END_REGION
END_ORGANIZATION_BLOCK

(* ===== HMI "HMI_RT_1" =====
system functions are stored by id; their names below are inferred from use
connection "HMI_Conexión_1": ETHERNET, SIMATIC S7 300/400 MPI

HMI tags "Tabla de variables estándar"
   "START_HMI" : Bool = PLC START_HMI AT %M3.7, 1 s
   "STOP_HMI" : Bool = PLC STOP_HMI AT %M4.0, 1 s
   "PE_HMI" : Bool = PLC PE_HMI AT %M4.1, 1 s
   "SEntrada" : Bool = PLC SEntrada AT %I1.1, 1 s
   "SPosDer1" : Bool = PLC SPosDer1 AT %I0.3, 1 s
   "SPosIzq1" : Bool = PLC SPosIzq1 AT %I0.2, 1 s
   "SPosDer2" : Bool = PLC SPosDer2 AT %I0.5, 1 s
   "SPosIzq2" : Bool = PLC SPosIzq2 AT %I0.7, 1 s
   "ClasificadorRecto" : Bool = PLC ClasificadorRecto AT %M4.4, 1 s
   "EnvVerde" : Bool = PLC EnvVerde AT %M4.3, 1 s
   "ClasificadorGiro" : Bool = PLC ClasificadorGiro AT %Q0.1, 1 s
   "EnvAzul" : Bool = PLC EnvAzul AT %M4.2, 1 s
   "SEntTapaVerd" : Bool = PLC SEntTapaVerd AT %I1.5, 1 s
   "SEntTapaAzul" : Bool = PLC SEntTapaAzul AT %I1.4, 1 s
   "SPoseDer3" : Bool = PLC SPoseDer3 AT %I0.6, 1 s
   "SPosIzq3" : Bool = PLC SPosIzq3 AT %I1.0, 1 s
   "ClampDere1" : Bool = PLC ClampDere1 AT %Q2.1, 1 s
   "ClampDere2" : Bool = PLC ClampDere2 AT %Q2.3, 1 s
   "SPosDer4" : Bool = PLC SPosDer4 AT %I1.3, 1 s
   "SPosIzq4" : Bool = PLC SPosIzq4 AT %I1.2, 1 s
   "VLlenadoEnvDer" : Bool = PLC VLlenadoEnvDer AT %Q1.3, 1 s
   "VLlenadoEnvIzq" : Bool = PLC VLlenadoEnvIzq AT %Q1.0, 1 s
   "ContadorEnvVerd" : Int = PLC ContadorEnvVerd AT %MW2, 1 s
   "MovZRDer" : Bool = PLC MovZRDer AT %Q2.7, 1 s
   "GrabRDer" : Bool = PLC GrabRDer AT %Q3.1, 1 s
   "ClampIzq1" : Bool = PLC ClampIzq1 AT %Q2.4, 1 s
   "MovZRIzq" : Bool = PLC MovZRIzq AT %Q3.2, 1 s
   "ClampIzq2" : Bool = PLC ClampIzq2 AT %Q2.6, 1 s
   "ContadorEnvAzul" : Int = PLC ContadorEnvAzul AT %MW0, 1 s

Template "Plantilla_1" 800x480
   Button "Start screen" at 1,2 size 78x58; TextOff 'Start screen'; PictureOff "NavigateHome_TP700_Comfort_TR"; PictureOn "NavigateHome_TP700_Comfort_TR"
      on Release: ActivateScreen("Imagen raíz", 0)
   Button "Template_Button" at 1,62 size 78x58; TextOff 'Text'
   Button "Template_Button_1" at 1,122 size 78x58; TextOff 'Text'
   Button "Template_Button_2" at 1,181 size 78x58; TextOff 'Text'
   Button "Template_Button_3" at 1,241 size 78x58; TextOff 'Text'
   Button "Template_Button_4" at 1,301 size 78x58; TextOff 'Text'
   Button "Log on" at 1,360 size 78x58; TextOff 'Log on'; PictureOff "Login_TP700_Comfort_TR"; PictureOn "Login_TP700_Comfort_TR"
      on Release: function_a2a04561()
   Button "Exit" at 1,420 size 78x58; TextOff 'Exit'; PictureOff "ExitRuntime_TP700_Comfort_TR"; PictureOn "ExitRuntime_TP700_Comfort_TR"
      on Release: StopRuntime(0)

screen "Imagen raíz" 800x480, template "Plantilla_1"
   GraphicView "Visor de gráficos_1" at 79,3 size 721x477; Picture "Gráfico_2"
   Button "Botón_1" at 219,276 size 118x50; TextOff 'INICIO / INICIAR'
      on Click: ActivateScreen("Principal", 0)
   TextField "Campo de texto_1" at 125,124 size 639x43; Text 'CLASIFICACIÓN, LLENADO Y TAPADO'
   TextField "Campo de texto_2" at 203,161 size 461x43; Text 'DE ENVASES DE PINTURAS'

screen "Principal" 800x480
   GraphicView "Visor de gráficos_5" at 317,129 size 177x74; Picture "Gráfico_1"
   Circle "Círculo_6" at 435,146 size 39x39
      Visibility <- "SPosIzq1"
   GraphicView "Visor de gráficos_4" at 243,281 size 254x75; Picture "Gráfico_1"
   Circle "Círculo_5" at 437,299 size 39x39
      Visibility <- "SPosDer1"
   SymbolLibrary "Librería de símbolos_14" at 430,257 size 57x61
   GraphicView "Visor de gráficos_9" at 502,50 size 150x75; Picture "Gráfico_1"
   SymbolLibrary "Librería de símbolos_1" at 332,15 size 92x106
   Slider "Deslizador_1" at 343,33 size 69x69; Caption 'AZUL'
   SymbolLibrary "Librería de símbolos_3" at 336,366 size 89x101
   Slider "Deslizador_2" at 347,382 size 69x69; Caption 'VERDE'
   GraphicView "Visor de gráficos_1" at 73,282 size 182x74; Picture "Gráfico_1"
   GraphicView "Visor de gráficos_2" at 176,129 size 151x141; Picture "Gráfico_3"
   GraphicView "Visor de gráficos_3" at 176,263 size 79x30; Picture "Gráfico_5"
   SymbolLibrary "Librería de símbolos_2" at 429,105 size 57x61
   GraphicView "Visor de gráficos_6" at 483,281 size 254x75; Picture "Gráfico_1"
   GraphicView "Visor de gráficos_7" at 482,129 size 254x74; Picture "Gráfico_1"
   GraphicView "Visor de gráficos_8" at 503,360 size 147x75; Picture "Gráfico_1"
   Button "Botón_1" at 56,82 size 84x36; TextOff 'STOP'
      on Press: SetBit("STOP_HMI")
      on Release: ResetBit("STOP_HMI")
   Button "Botón_2" at 56,29 size 84x36; TextOff 'START'
      on Press: SetBit("START_HMI")
      on Release: ResetBit("START_HMI")
   Circle "Círculo_1" at 517,377 size 39x39
      Visibility <- "SEntTapaVerd"
   Circle "Círculo_2" at 514,67 size 39x39
      Visibility <- "SEntTapaAzul"
   Switch "Interruptor_1" at 31,133 size 136x60; CaptionText 'PARADA EMERG'; TextOff 'OFF'; TextOn 'ON'
      on SwitchOn: SetBit("PE_HMI")
      on SwitchOff: ResetBit("PE_HMI")
   Circle "Círculo_3" at 599,298 size 39x39
      Visibility <- "SPosDer2"
   Circle "Círculo_4" at 597,146 size 39x39
      Visibility <- "SPosIzq2"
   Circle "Círculo_7" at 89,298 size 39x39
      Visibility <- "SEntrada"
   GraphicView "Visor de gráficos_10" at 158,323 size 142x69; Picture "Clasif-removebg-preview"
      Visibility <- "ClasificadorRecto"
   Circle "Círculo_8" at 194,298 size 39x39
      Visibility <- "EnvVerde"
   GraphicView "Visor de gráficos_11" at 171,279 size 99x95; Picture "Clasfi2-removebg-preview"
      Visibility <- "ClasificadorGiro"
   Circle "Círculo_9" at 195,275 size 39x39
      Visibility <- "EnvAzul"
   Circle "Círculo_10" at 599,377 size 39x39
      Visibility <- "SPoseDer3"
   Circle "Círculo_11" at 597,67 size 39x39
      Visibility <- "SPosIzq3"
   Rectangle "Rectángulo_3" at 638,359 size 11x72
      Visibility <- "ClampDere2"
   Rectangle "Rectángulo_4" at 585,359 size 64x11
      Visibility <- "ClampDere2"
   Rectangle "Rectángulo_5" at 588,280 size 64x11
      Visibility <- "ClampDere1"
   Rectangle "Rectángulo_6" at 641,281 size 11x71
      Visibility <- "ClampDere1"
   Rectangle "Rectángulo_7" at 638,376 size 11x55
      Visibility <- "ClampDere2"
   Circle "Círculo_12" at 599,386 size 39x39
      Visibility <- "ClampDere2"
   Rectangle "Rectángulo_8" at 585,375 size 64x11
      Visibility <- "ClampDere2"
   Rectangle "Rectángulo_9" at 641,297 size 11x55
      Visibility <- "ClampDere1"
   Rectangle "Rectángulo_10" at 587,295 size 64x11
      Visibility <- "ClampDere1"
   Circle "Círculo_13" at 599,307 size 39x39
      Visibility <- "SPosDer2"
   Circle "Círculo_14" at 667,299 size 39x39
      Visibility <- "SPosDer4"
   Rectangle "Rectángulo_11" at 452,275 size 6x48
      Visibility <- "VLlenadoEnvDer"
   Circle "Círculo_15" at 666,146 size 39x39
      Visibility <- "SPosIzq4"
   Rectangle "Rectángulo_12" at 451,121 size 6x48
      Visibility <- "VLlenadoEnvIzq"
   IOField "Campo ES_1" at 694,403 size 64x32; FormatPattern 9999
      ProcessValue <- "ContadorEnvVerd"
   TextField "Campo de texto_1" at 679,365 size 100x22; Text 'N° Evanses'
   TextField "Campo de texto_2" at 695,380 size 63x22; Text 'Verdes'
   Rectangle "Rectángulo_14" at 607,396 size 22x62
      Visibility <- "MovZRDer"
   Circle "Círculo_16" at 600,306 size 39x39
      Visibility <- "MovZRDer"
   Rectangle "Rectángulo_16" at 607,318 size 22x140
      Visibility <- "MovZRDer"
   Rectangle "Rectángulo_15" at 636,134 size 11x54
      Visibility <- "ClampIzq1"
   Rectangle "Rectángulo_17" at 583,177 size 64x11
      Visibility <- "ClampIzq1"
   Rectangle "Rectángulo_18" at 637,133 size 11x71
      Visibility <- "ClampIzq1"
   Rectangle "Rectángulo_19" at 584,193 size 64x11
      Visibility <- "ClampIzq1"
   Rectangle "Rectángulo_20" at 636,54 size 11x55
      Visibility <- "ClampIzq2"
   Circle "Círculo_18" at 597,138 size 39x39
      Visibility <- "SPosIzq2"
   Circle "Círculo_19" at 598,139 size 39x39
      Visibility <- "MovZRIzq"
   Rectangle "Rectángulo_21" at 583,98 size 64x11
      Visibility <- "ClampIzq2"
   Circle "Círculo_17" at 597,60 size 39x39
      Visibility <- "ClampIzq2"
   Rectangle "Rectángulo_22" at 583,114 size 64x11
      Visibility <- "ClampIzq2"
   Rectangle "Rectángulo_23" at 636,54 size 11x71
      Visibility <- "ClampIzq2"
   Rectangle "Rectángulo_25" at 605,26 size 22x62
      Visibility <- "MovZRIzq"
   Rectangle "Rectángulo_26" at 605,26 size 22x140
      Visibility <- "MovZRIzq"
   IOField "Campo ES_2" at 693,82 size 64x32; FormatPattern 9999
      ProcessValue <- "ContadorEnvAzul"
   TextField "Campo de texto_3" at 678,44 size 100x22; Text 'N° Evanses'
   TextField "Campo de texto_4" at 699,59 size 60x22; Text 'Azules'
   Button "Botón_3" at 17,426 size 85x38; TextOff 'MENU'
      on Click: ActivateScreen("Imagen raíz", 0)
*)